// SIMATIC S7-200 project (STEP 7-Micro/WIN), CPU 224XP REL 02.01

SYMBOL_TABLE 全局符号表
急停按钮             I0.0     // I0.0
喷涂输送             I0.1     // I0.1
喷涂真空             I0.2     // I0.2
隔膜泵              I0.3     // I0.3
喷涂加热             I0.4     // I0.4
流平输送             I0.5     // I0.5
流平加热             I0.6     // I0.6
干燥输送I            I0.7     // I0.7
一灯               I1.0     // I1.0
一灯强              I1.1     // I1.1
二灯               I1.2     // I1.2
二灯强              I1.3     // I1.3
三灯               I1.4     // I1.4
四灯               I1.5     // I1.5
喷涂异常             I2.0     // i2.0
真空异常             I2.1     // i2.1
流平异常             I2.2     // i2.2
干燥异常             I2.3     // i2.3
风机1异常            I2.4     // i2.4
风机2异常            I2.5     // i2.5
安全门1异常           I2.6     // i2.6
安全门2异常           I2.7     // i2.7
喷涂输送Q            Q0.0     // Q0.0
真空Q              Q0.1     // Q0.1
流平输送Q            Q0.2     // Q0.2
干燥输送Q            Q0.3     // Q0.3
一灯Q              Q0.4     // Q0.4
一灯强Q             Q0.5     // Q0.5
二灯Q              Q0.6     // Q0.6
二灯强Q             Q0.7     // Q0.7
三灯Q              Q1.0     // Q1.0
四灯Q              Q1.1     // Q1.1
喷涂加热Q            Q2.0     // Q2.0
流平加热Q            Q2.1     // Q2.1
风机1Q             Q2.2     // Q2.2
风机2Q             Q2.3     // Q2.3
电磁阀              Q2.4     // Q2.4
红色灯              Q2.5     // Q2.5
绿色灯              Q2.6     // Q2.6
黄色灯              Q2.7     // Q2.7
一灯电流             AIW4     // AIW4
二灯电流             AIW6     // AIW6
三灯电流             AIW8     // AIW8
四灯电流             AIW10    // AIW10
喷涂温度             AIW12    // AIW12
流平温度             AIW14    // AIW14
干燥温度             AIW16    // AIW16
真空速度             AQW0     // AQW0
流平速度             AQW2     // AQW2
干燥速度             AQW4     // AQW4
灯1电流             VD0      // VD0
灯2电流             VD2      // VD2
灯3电流             VD4      // VD4
灯4电流             VD6      // VD6
温度喷涂             VD8      // VD8
温度流平             VD10     // VD10
温度干燥             VD12     // VD12
真空速度给定           VD14     // VD14
流平速度给定           VD16     // VD16
干燥速度给定           VD18     // VD18
急停状态             M0.0     // M0.0
安全门1             M0.1     // M0.1
安全门2             M0.2     // M0.2
安全门              M0.3     // M0.3
始终ON             SM0.0    // SM0.0
喷涂上限             VD20     // VD20
喷涂下限             VD22     // VD22
流平上限             VD24     // VD24
流平下限             VD26     // VD26
干燥上限             VD28     // VD28
干燥下限             VD30     // VD30
干燥极限             VD32     // VD32
风机开启             VD34     // VD34
风机关闭             VD36     // VD36
一灯过流             VD40     // VD40
二灯过流             VD42     // VD42
三灯过流             VD44     // VD44
四灯过流             VD48     // VD48
真空变频异常           M0.4     // M0.4
喷涂输送异常           M0.5     // M0.5
流平输送异常           M0.6     // M0.6
干燥输送异常           M0.7     // M0.7
散热风机异常           M1.0     // M1.0
干燥风机异常           M1.1     // M1.1
干燥加热控制           M1.2     // M1.2
一过流              M1.4     // M1.4
二过流              M1.5     // M1.5
三过流              M1.6     // M1.6
四过流              M1.7     // M1.7
故障复位             M2.0     // M2.0
风机控制             M1.3     // M1.3
END_SYMBOL_TABLE

ORGANIZATION_BLOCK 主程序:OB1
TITLE=主程序
BEGIN
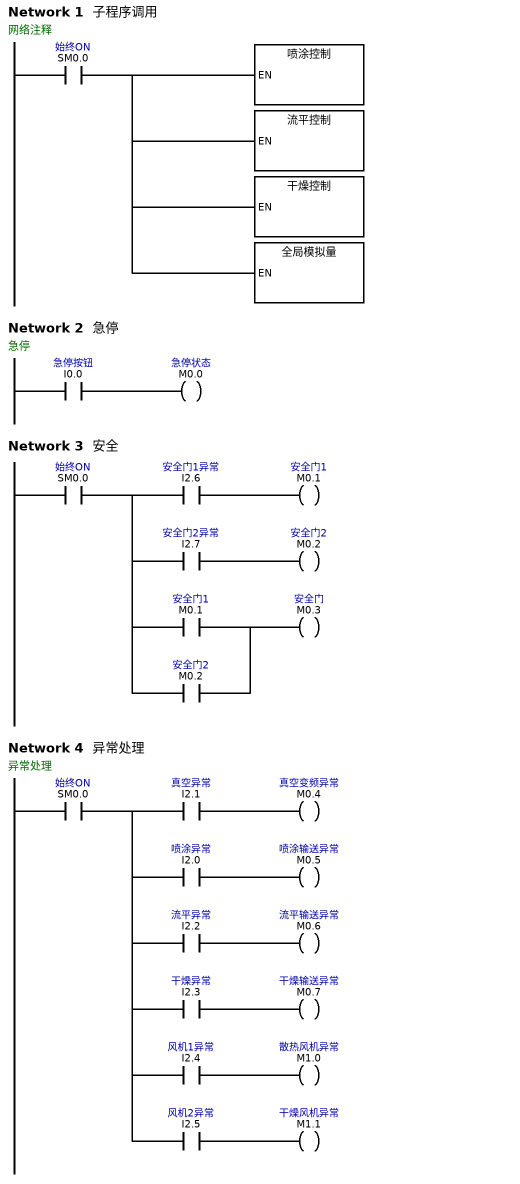
Network 1 // 子程序调用
// 网络注释
LD     始终ON:SM0.0
CALL   喷涂控制:SBR0
CALL   流平控制:SBR1
CALL   干燥控制:SBR2
CALL   全局模拟量:SBR3
Network 2 // 急停
// 急停
LD     急停按钮:I0.0
=      急停状态:M0.0
Network 3 // 安全
LD     始终ON:SM0.0
LPS
A      安全门1异常:I2.6
=      安全门1:M0.1
LRD
A      安全门2异常:I2.7
=      安全门2:M0.2
LPP
LD     安全门1:M0.1
O      安全门2:M0.2
ALD
=      安全门:M0.3
Network 4 // 异常处理
// 异常处理
LD     始终ON:SM0.0
LPS
A      真空异常:I2.1
=      真空变频异常:M0.4
LRD
A      喷涂异常:I2.0
=      喷涂输送异常:M0.5
LRD
A      流平异常:I2.2
=      流平输送异常:M0.6
LRD
A      干燥异常:I2.3
=      干燥输送异常:M0.7
LRD
A      风机1异常:I2.4
=      散热风机异常:M1.0
LPP
A      风机2异常:I2.5
=      干燥风机异常:M1.1
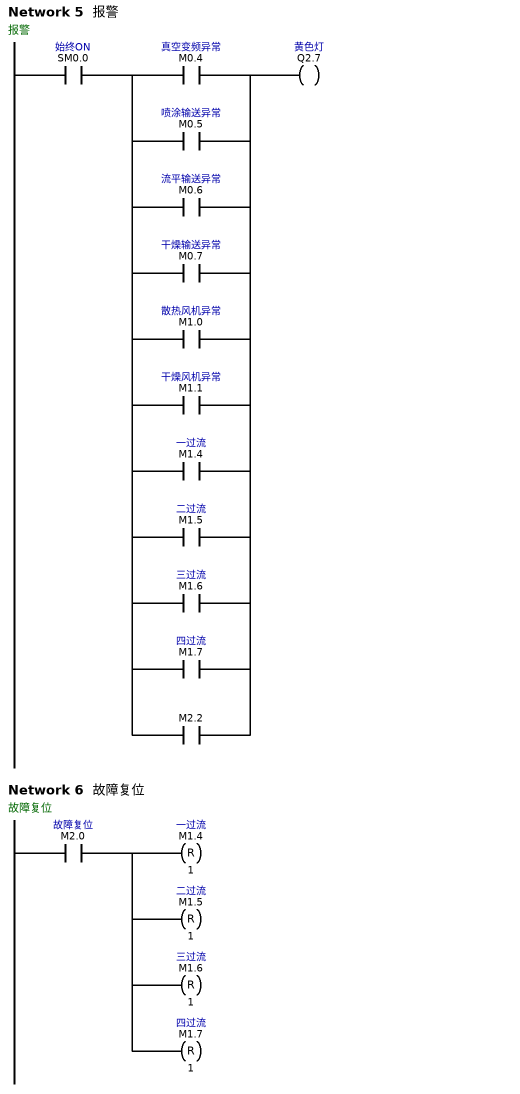
Network 5 // 报警
// 报警
LD     始终ON:SM0.0
LD     真空变频异常:M0.4
O      喷涂输送异常:M0.5
O      流平输送异常:M0.6
O      干燥输送异常:M0.7
O      散热风机异常:M1.0
O      干燥风机异常:M1.1
O      一过流:M1.4
O      二过流:M1.5
O      三过流:M1.6
O      四过流:M1.7
O      M2.2
ALD
=      黄色灯:Q2.7
Network 6 // 故障复位
// 故障复位
LD     故障复位:M2.0
R      一过流:M1.4, 1
R      二过流:M1.5, 1
R      三过流:M1.6, 1
R      四过流:M1.7, 1
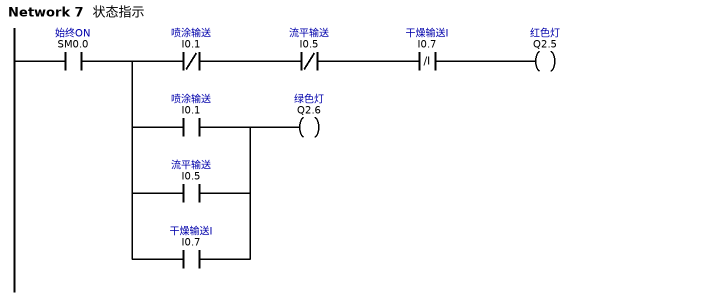
Network 7 // 状态指示
LD     始终ON:SM0.0
LPS
AN     喷涂输送:I0.1
AN     流平输送:I0.5
ANI    干燥输送I:I0.7
=      红色灯:Q2.5
LPP
LD     喷涂输送:I0.1
O      流平输送:I0.5
O      干燥输送I:I0.7
ALD
=      绿色灯:Q2.6
END_ORGANIZATION_BLOCK

SUBROUTINE_BLOCK 喷涂控制:SBR0
TITLE=子程序注释
BEGIN
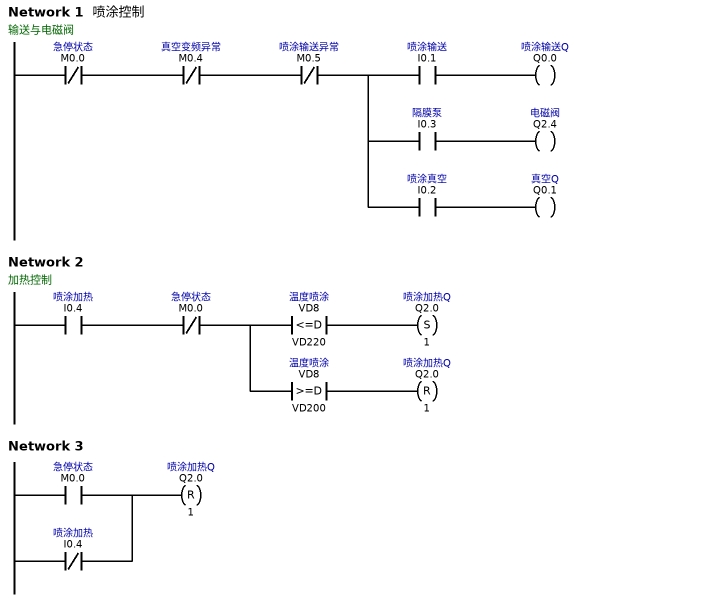
Network 1 // 喷涂控制
// 输送与电磁阀
LDN    急停状态:M0.0
AN     真空变频异常:M0.4
AN     喷涂输送异常:M0.5
LPS
A      喷涂输送:I0.1
=      喷涂输送Q:Q0.0
LRD
A      隔膜泵:I0.3
=      电磁阀:Q2.4
LPP
A      喷涂真空:I0.2
=      真空Q:Q0.1
Network 2
// 加热控制
LD     喷涂加热:I0.4
AN     急停状态:M0.0
LPS
AD<=   温度喷涂:VD8, VD220
S      喷涂加热Q:Q2.0, 1
LPP
AD>=   温度喷涂:VD8, VD200
R      喷涂加热Q:Q2.0, 1
Network 3
LD     急停状态:M0.0
ON     喷涂加热:I0.4
R      喷涂加热Q:Q2.0, 1
END_SUBROUTINE_BLOCK

SUBROUTINE_BLOCK 流平控制:SBR1
TITLE=子程序注释
BEGIN
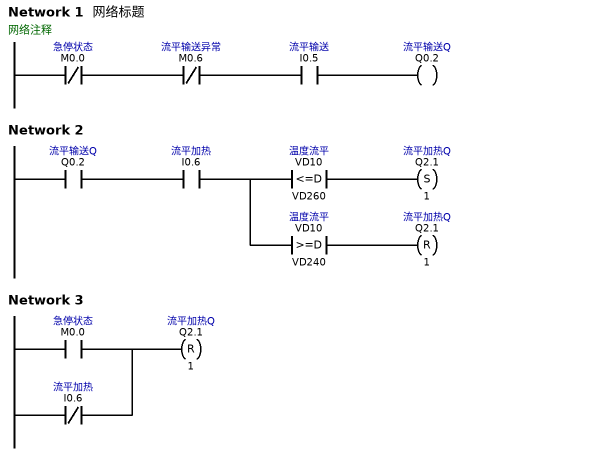
Network 1 // 网络标题
// 网络注释
LDN    急停状态:M0.0
AN     流平输送异常:M0.6
A      流平输送:I0.5
=      流平输送Q:Q0.2
Network 2
LD     流平输送Q:Q0.2
A      流平加热:I0.6
LPS
AD<=   温度流平:VD10, VD260
S      流平加热Q:Q2.1, 1
LPP
AD>=   温度流平:VD10, VD240
R      流平加热Q:Q2.1, 1
Network 3
LD     急停状态:M0.0
ON     流平加热:I0.6
R      流平加热Q:Q2.1, 1
END_SUBROUTINE_BLOCK

SUBROUTINE_BLOCK 干燥控制:SBR2
TITLE=子程序注释
BEGIN
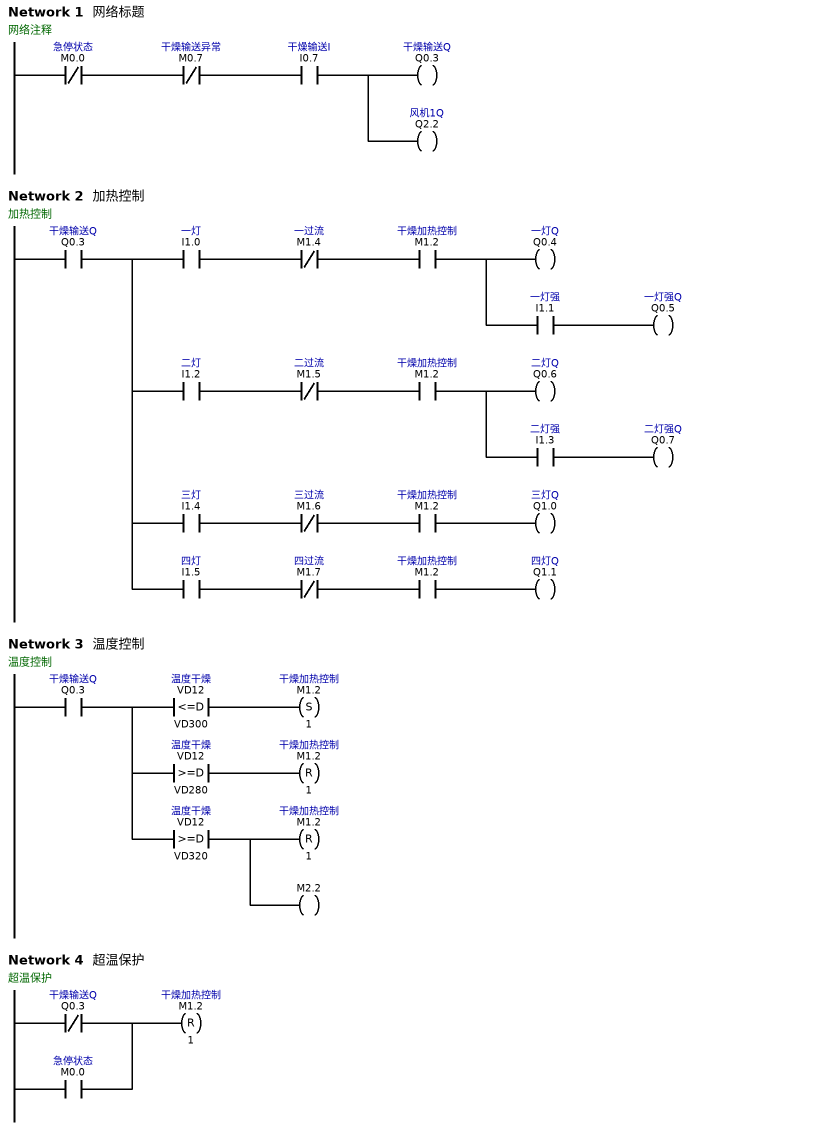
Network 1 // 网络标题
// 网络注释
LDN    急停状态:M0.0
AN     干燥输送异常:M0.7
A      干燥输送I:I0.7
=      干燥输送Q:Q0.3
=      风机1Q:Q2.2
Network 2 // 加热控制
// 加热控制
LD     干燥输送Q:Q0.3
LPS
A      一灯:I1.0
AN     一过流:M1.4
A      干燥加热控制:M1.2
=      一灯Q:Q0.4
A      一灯强:I1.1
=      一灯强Q:Q0.5
LRD
A      二灯:I1.2
AN     二过流:M1.5
A      干燥加热控制:M1.2
=      二灯Q:Q0.6
A      二灯强:I1.3
=      二灯强Q:Q0.7
LPP
LPS
A      三灯:I1.4
AN     三过流:M1.6
A      干燥加热控制:M1.2
=      三灯Q:Q1.0
LPP
A      四灯:I1.5
AN     四过流:M1.7
A      干燥加热控制:M1.2
=      四灯Q:Q1.1
Network 3 // 温度控制
// 温度控制
LD     干燥输送Q:Q0.3
LPS
AD<=   温度干燥:VD12, VD300
S      干燥加热控制:M1.2, 1
LRD
AD>=   温度干燥:VD12, VD280
R      干燥加热控制:M1.2, 1
LPP
AD>=   温度干燥:VD12, VD320
R      干燥加热控制:M1.2, 1
=      M2.2
Network 4 // 超温保护
// 超温保护
LDN    干燥输送Q:Q0.3
O      急停状态:M0.0
R      干燥加热控制:M1.2, 1
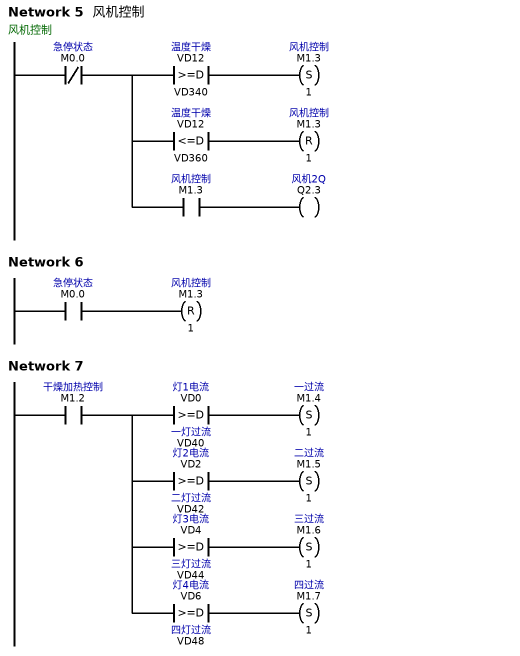
Network 5 // 风机控制
// 风机控制
LDN    急停状态:M0.0
LPS
AD>=   温度干燥:VD12, VD340
S      风机控制:M1.3, 1
LRD
AD<=   温度干燥:VD12, VD360
R      风机控制:M1.3, 1
LPP
A      风机控制:M1.3
=      风机2Q:Q2.3
Network 6
LD     急停状态:M0.0
R      风机控制:M1.3, 1
Network 7
LD     干燥加热控制:M1.2
LPS
AD>=   灯1电流:VD0, 一灯过流:VD40
S      一过流:M1.4, 1
LRD
AD>=   灯2电流:VD2, 二灯过流:VD42
S      二过流:M1.5, 1
LRD
AD>=   灯3电流:VD4, 三灯过流:VD44
S      三过流:M1.6, 1
LPP
AD>=   灯4电流:VD6, 四灯过流:VD48
S      四过流:M1.7, 1
END_SUBROUTINE_BLOCK

SUBROUTINE_BLOCK 全局模拟量:SBR3
TITLE=子程序注释
BEGIN
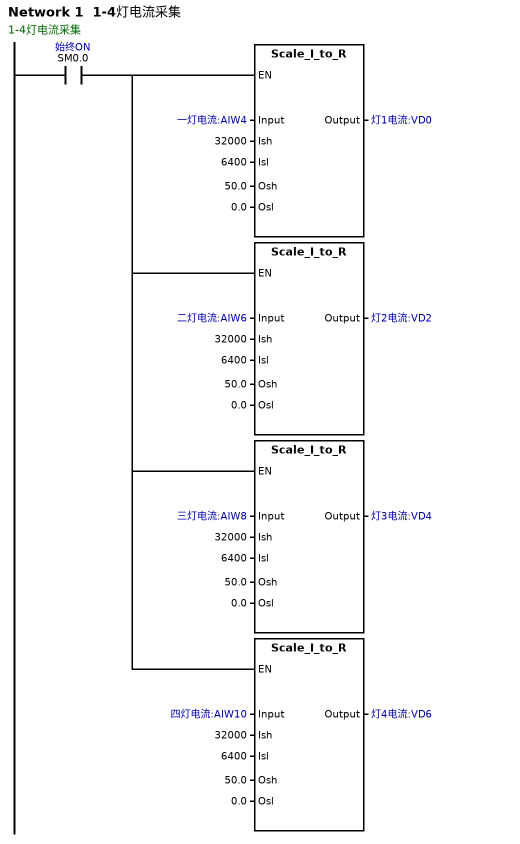
Network 1 // 1-4灯电流采集
// 1-4灯电流采集
LD     始终ON:SM0.0
CALL   Scale_I_to_R:SBR4, 一灯电流:AIW4, 32000, 6400, 50.0, 0.0, 灯1电流:VD0
CALL   Scale_I_to_R:SBR4, 二灯电流:AIW6, 32000, 6400, 50.0, 0.0, 灯2电流:VD2
CALL   Scale_I_to_R:SBR4, 三灯电流:AIW8, 32000, 6400, 50.0, 0.0, 灯3电流:VD4
CALL   Scale_I_to_R:SBR4, 四灯电流:AIW10, 32000, 6400, 50.0, 0.0, 灯4电流:VD6
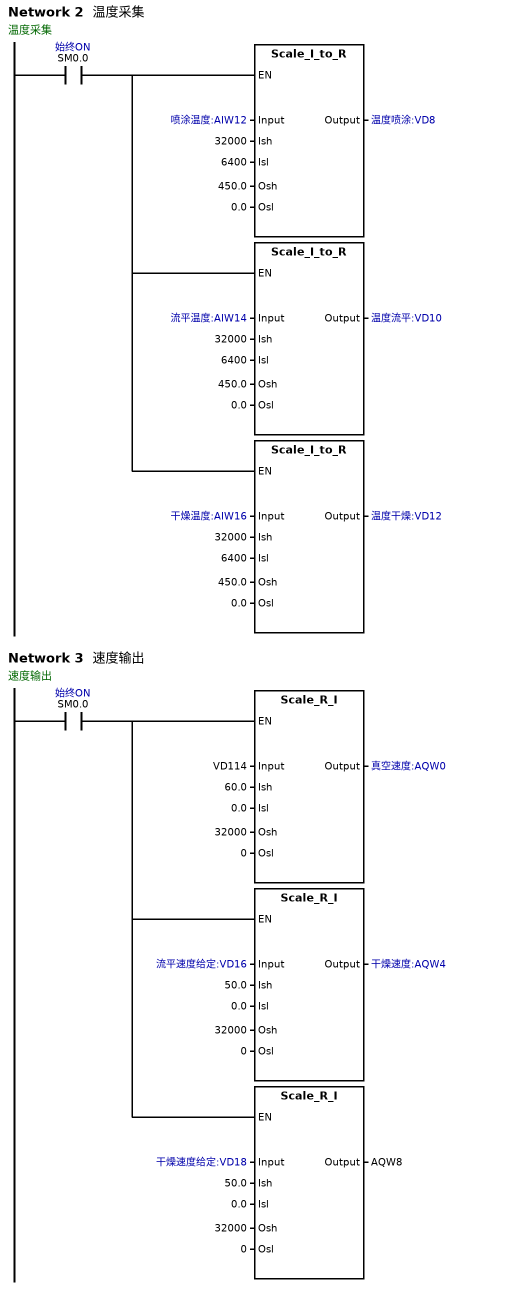
Network 2 // 温度采集
// 温度采集
LD     始终ON:SM0.0
CALL   Scale_I_to_R:SBR4, 喷涂温度:AIW12, 32000, 6400, 450.0, 0.0, 温度喷涂:VD8
CALL   Scale_I_to_R:SBR4, 流平温度:AIW14, 32000, 6400, 450.0, 0.0, 温度流平:VD10
CALL   Scale_I_to_R:SBR4, 干燥温度:AIW16, 32000, 6400, 450.0, 0.0, 温度干燥:VD12
Network 3 // 速度输出
// 速度输出
LD     始终ON:SM0.0
CALL   Scale_R_I:SBR5, VD114, 60.0, 0.0, 32000, 0, 真空速度:AQW0
CALL   Scale_R_I:SBR5, 流平速度给定:VD16, 50.0, 0.0, 32000, 0, 干燥速度:AQW4
CALL   Scale_R_I:SBR5, 干燥速度给定:VD18, 50.0, 0.0, 32000, 0, AQW8
END_SUBROUTINE_BLOCK

// SBR4: protected block, not included

// SBR5: protected block, not included
